{attribute 'GeneratedUsingTerminal: EL7041-1000-0021'}
{attribute addProperty BoxType "EL7041-1000-0021"}
{attribute addProperty Id "AdsAddrAT %I*TcoIo.TcoAmsAddr0Chn0AT %I*USINT1StateAT %I*UINT2"}
{attribute addProperty CRC "3574367557"}
{attribute addProperty Size "3"}
TYPE InfoData_D50C8545 EXTENDS TcoIo.InputBase_8311D824 :
STRUCT
	{attribute addProperty Name "AdsAddr"}
	AdsAddr AT %I* : TcoIo.TcoAmsAddr;
	{attribute addProperty Name "Chn0"}
	Chn0 AT %I* : USINT;
	{attribute addProperty Name "State"}
	State AT %I* : UINT;
END_STRUCT
END_TYPE

(* stored: Version 1.2.0.0, ProductVersion 3.1.4024.11
   DUT InfoData_D50C8545: Id {e261cbfc-0afa-03dd-2628-57d1490197e4} *)
